// TIA Portal V20 export
// export: Created 2025-12-01T14:56:12.0238865Z, ExportSetting None, DisplayName Totally Integrated Automation Portal, DisplayVersion V20 Update 3, DisplayName TIA Portal Openness, DisplayVersion V20 Update 3, DisplayName TIA Portal Version Control Interface, DisplayVersion V20 Update 3, DisplayName STEP 7 Professional, DisplayVersion V20 Update 3, DisplayName STEP 7 Safety, DisplayVersion V20 Update 2, DisplayName WinCC Basic/Comfort/Advanced, DisplayVersion V20 Update 3, DisplayName WinCC Professional, DisplayVersion V20 Update 3, DisplayName WinCC Unified, DisplayVersion V20 Update 3
TYPE "InternasDeLaZona"
   STRUCT
      MesasParo : Bool;
      MesasManual : Bool;
      MesasBlando : Bool;
      MesasError : Bool;
      MesasTodasParo : Bool;
      MesasTodasManual : Bool;
      Libre_06 : Bool;
      Libre_07 : Bool;
      Libre_10 : Bool;
      Libre_11 : Bool;
      Libre_12 : Bool;
      Libre_13 : Bool;
      Libre_14 : Bool;
      BalizaRoja : Bool;
      BalizaNaranja : Bool;
      BalizaVerde : Bool;
   END_STRUCT;
END_TYPE
